TYPE "Button_Class"
VERSION : 0.1
   STRUCT
      state : Bool;
      light : Bool;
      p : Bool;
   END_STRUCT;

END_TYPE

